{attribute 'qualified_only'}
{attribute 'strict'}
{attribute 'to_string'}
TYPE SignalStatusLampStatus_t :
(
	NONE := 0,
	OPERATIONAL := 1,
	WARNING := 2,
	ERROR := 3,
	STARTING := 4,
	STOPPING := 5
);
END_TYPE

(* stored: Version 1.1.0.1
   EnumerationTextList SignalStatusLampStatus_t: Id {06b60611-4eb0-4e35-ad51-df477db9c76d} *)
